FUNCTION_BLOCK FB_ejemplo_Propiedad
VAR_INPUT
END_VAR
VAR_OUTPUT
END_VAR
VAR_IN_OUT
	myIN_OUT : INT;
END_VAR
VAR
	myBool : BOOL;
	myInt : INT;
	myST  : ST_Property;
END_VAR

PROPERTY Value_INT_OUT : INT
GET
IF NOT __ISVALIDREF(myIN_OUT) THEN
	RETURN;
END_IF

Value_INT_OUT := myIN_OUT;
END_GET
SET
myIN_OUT := Value_INT_OUT;
END_SET
END_PROPERTY

PROPERTY ValueBool : BOOL
GET
ValueBool := myBool;
END_GET
SET
 myBool := ValueBool;
END_SET
END_PROPERTY

PROPERTY ValueInt : INT
GET
ValueInt := myint;
END_GET
SET
 myint := ValueInt;
END_SET
END_PROPERTY

PROPERTY ValueST : reference to ST_Property
GET
ValueST REF= myST;
END_GET
SET
IF NOT __ISVALIDREF(myIN_OUT) THEN
	RETURN;
END_IF

myST := ValueST;
END_SET
END_PROPERTY

END_FUNCTION_BLOCK

(* stored: Version 1.1.0.1, ProductVersion 3.1.4024.12
   POU FB_ejemplo_Propiedad: Id {53403d56-6301-4aee-9142-b3bd61d2b285}, SpecialFunc None
   Property Value_INT_OUT: Id {74661cd1-1310-4f4c-b576-728ac27ce460}
   Get Get: Id {0b4ba3a1-227e-48ae-ba4b-b1dee639a238}
   Set Set: Id {0a819901-1711-49d1-99ba-703d67b1f949}
   Property ValueBool: Id {e79b1ae8-d8e8-4277-9ceb-b086c5c3097a}
   Get Get: Id {717513e8-d69b-48df-8f15-0ae7c6ffedc5}
   Set Set: Id {80c164f1-a865-4312-8c5f-9be5079c21f9}
   Property ValueInt: Id {133670a7-09af-415f-957f-31103a022050}
   Get Get: Id {99e3d0a0-07d5-4640-874f-35fdef4875fa}
   Set Set: Id {2aa76308-b9d0-4df7-abc3-5933a1c4c6ee}
   Property ValueST: Id {363a33a0-bfc3-42f4-861a-12e4c4928f01}
   Get Get: Id {881eebdf-89d5-4979-a45d-62e550b19232}
   Set Set: Id {2fe34d5e-d91e-450b-9a12-99f8521f55c9} *)
